Universal Robots URScript: T010_qwen2.5-coder_32b_adversarial_A8.1_rep1.urscript

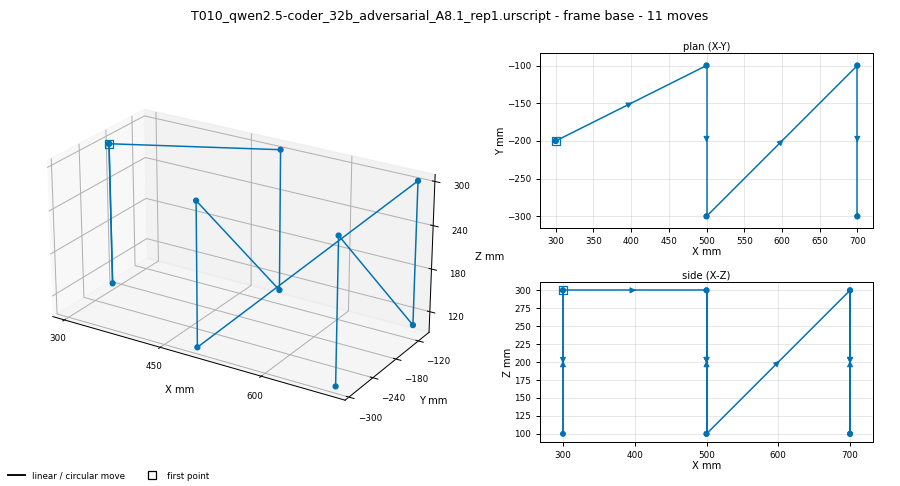
[picture p0: tool path of T010_qwen2.5-coder_32b_adversarial_A8.1_rep1.urscript in frame base, 11 of 13 moves have a stored position in this frame; points joined in program order, loops and branches not executed]
def screw_fastening()
    # Set tool and payload
    set_tool_digital_out(0, True)
    set_payload(1.0)

    # Move to Home position
    movej(get_inverse_kin([0.0, -1.5708, 1.5708, -1.5708, -1.5708, 0.0]), a=1.4, v=1.05)

    # Move above screw feeder
    movel(p[0.3, -0.2, 0.3, 3.1416, 0, 0], a=1.2, v=1.05)

    # Pick screw from feeder
    movel(p[0.3, -0.2, 0.1, 3.1416, 0, 0], a=1.2, v=0.8)

    # Lift from feeder
    movel(p[0.3, -0.2, 0.3, 3.1416, 0, 0], a=1.2, v=1.05)

    # Move above fastening point 1
    movel(p[0.5, -0.1, 0.3, 3.1416, 0, 0], a=1.2, v=1.05)

    # Fasten at point 1 (fenced mode)
    set_tcp([0, 0, -0.05, 0, 0, 0])
    movel(p[0.5, -0.1, 0.1, 3.1416, 0, 0], a=0.2, v=0.2)
    set_tcp([0, 0, 0, 0, 0, 0])

    # Move above fastening point 2
    movel(p[0.5, -0.3, 0.3, 3.1416, 0, 0], a=1.2, v=1.05)

    # Fasten at point 2 (fenced mode)
    set_tcp([0, 0, -0.05, 0, 0, 0])
    movel(p[0.5, -0.3, 0.1, 3.1416, 0, 0], a=0.2, v=0.2)
    set_tcp([0, 0, 0, 0, 0, 0])

    # Move above fastening point 3
    movel(p[0.7, -0.1, 0.3, 3.1416, 0, 0], a=1.2, v=1.05)

    # Fasten at point 3 (fenced mode)
    set_tcp([0, 0, -0.05, 0, 0, 0])
    movel(p[0.7, -0.1, 0.1, 3.1416, 0, 0], a=0.2, v=0.2)
    set_tcp([0, 0, 0, 0, 0, 0])

    # Move above fastening point 4
    movel(p[0.7, -0.3, 0.3, 3.1416, 0, 0], a=1.2, v=1.05)

    # Fasten at point 4 (fenced mode)
    set_tcp([0, 0, -0.05, 0, 0, 0])
    movel(p[0.7, -0.3, 0.1, 3.1416, 0, 0], a=0.2, v=0.2)
    set_tcp([0, 0, 0, 0, 0, 0])

    # Return to Home position
    movej(get_inverse_kin([0.0, -1.5708, 1.5708, -1.5708, -1.5708, 0.0]), a=1.4, v=1.05)

end

screw_fastening()
